# B&R Automation Studio project laba2
Automation Studio 4.5.2.102

## Configuration MainConfig

### Task classes (Cpu.sw)
```
Cyclic#1 (cycle 2000 us, tolerance 0 us):
  ncsdcctrl <- ncsdcctrl.prg
Cyclic#3:
  Program <- Program.prg
DataObjects: Acp10sys
NcDataObjects: acp10etxen <- acp10etxen.dob, gAxis01a <- gAxis01obj.gAxis01a.dob, gAxis01i <- gAxis01obj.gAxis01i.dob
Binaries: TCData, udbdef, ashwd, Role, User, sysconf, ashwac, asfw, arconfig, iomap, Acp10map, acp10cfg
Libraries: Acp10sdc [disabled], sys_lib, Runtime, asstring, Acp10man, Acp10par, NcGlobal, Acp10_MC, brsystem, AsBrStr, DriveLib, astime, fileio, powerlnk, asieccon
```

### Hardware
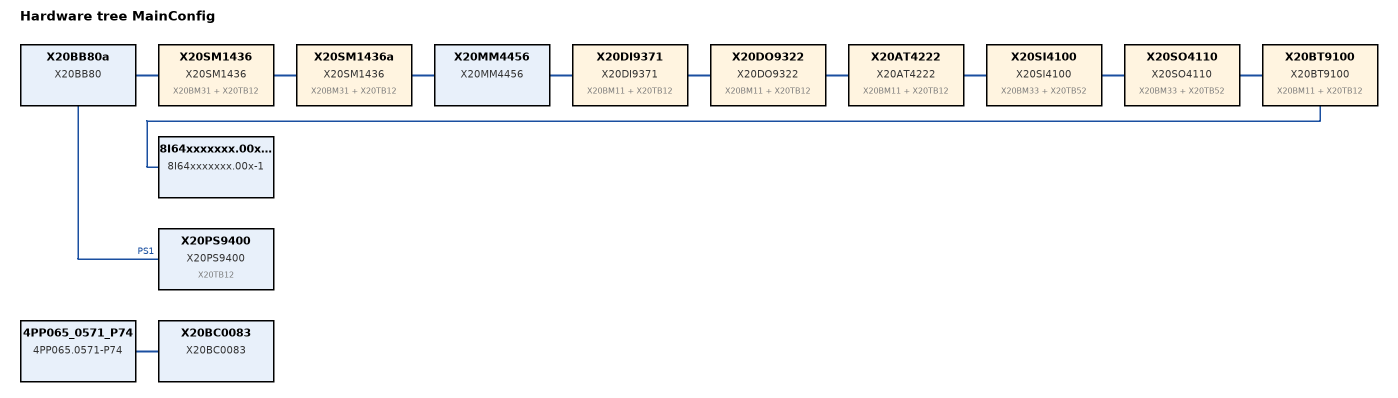
```
4PP065_0571_P74 : 4PP065.0571-P74 v1.1.2.0
  Connector IF4:
    InaNodeNumber = 1
  Connector IF5:
    ActivateDevice = 1
    Mode = Manual
    InternetAddress = 10.0.1.11
    SubnetMask = 255.255.255.0
  ConfigurationID = labBR
  TimerDeviceType = EPLX2X
  TimerDevice = 4PP065_0571_P74.IF4
  TaskClassIdleTime = 2000
  Cyclic1Duration = 2000
  Cyclic1Tolerance = 0
  Cyclic1Output = 1
8I64xxxxxxx.00x-1 : 8I64xxxxxxx.00x-1 v1.3.9.1  [X2X1 -> X20BT9100.X2X1 [Cable Type=X2XCable, Length=10, Version=1.0.0.2]]
  FunctionModel = Standard
  packedETAD = packed
  packedETI = packed
  packedCMDD = packed
  packedCMI = packed
  UNS = 220
  NCR = 10
  NSP = 890
  COS = 64
  RSC = 33000
X20AT4222 : X20AT4222 v1.2.3.0  [SS1 -> X20TB12e.SS; SL -> X20BM11c.SL1]
X20BB80a : X20BB80 v1.0.2.0
X20BC0083 : X20BC0083 v2.14.0.0  [PLK1 -> 4PP065_0571_P74.IF4 (NodeNumber=2) [Cable Type=PowerlinkCable, Length=10, Version=1.0.0.2]; SL -> X20BB80a.SL1]
X20BM11 : X20BM11 v1.0.0.1  [X2X1 -> X20BM33a.X2X2]
X20BM11a : X20BM11 v1.0.0.1  [X2X1 -> X20MM4456.X2X2]
X20BM11b : X20BM11 v1.0.0.1  [X2X1 -> X20BM11a.X2X2]
X20BM11c : X20BM11 v1.0.0.1  [X2X1 -> X20BM11b.X2X2]
X20BM31 : X20BM31 v1.0.0.1  [X2X1 -> X20BB80a.IF1]
X20BM31a : X20BM31 v1.0.0.1  [X2X1 -> X20BM31.X2X2]
X20BM33 : X20BM33 v1.0.0.4  [X2X1 -> X20BM11c.X2X2]
X20BM33a : X20BM33 v1.0.0.4  [X2X1 -> X20BM33.X2X2]
X20BT9100 : X20BT9100 v1.0.3.0  [SS1 -> X20TB12f.SS; SL -> X20BM11.SL1]
X20DI9371 : X20DI9371 v1.0.2.0  [SS1 -> X20TB12c.SS; SL -> X20BM11a.SL1]
X20DO9322 : X20DO9322 v1.0.3.0  [SS1 -> X20TB12d.SS; SL -> X20BM11b.SL1]
X20MM4456 : X20MM4456 v1.4.0.0  [X2X1 -> X20BM31a.X2X2]
X20PS9400 : X20PS9400 v1.0.2.4  [SS1 -> X20TB12.SS; PS -> X20BB80a.PS1]
X20SI4100 : X20SI4100 v1.10.1.1  [SS1 -> X20TB52.SS; SL -> X20BM33.SL1]
X20SM1436 : X20SM1436 v2.3.0.0  [SS1 -> X20TB12a.SS; SL -> X20BM31.SL1]
X20SM1436a : X20SM1436 v2.3.0.0  [SS1 -> X20TB12b.SS; SL -> X20BM31a.SL1]
X20SO4110 : X20SO4110 v1.10.1.1  [SS1 -> X20TB52a.SS; SL -> X20BM33a.SL1]
  SafeModuleID = 3
X20TB12 : X20TB12 v1.0.0.0
X20TB12a : X20TB12 v1.0.0.0
X20TB12b : X20TB12 v1.0.0.0
X20TB12c : X20TB12 v1.0.0.0
X20TB12d : X20TB12 v1.0.0.0
X20TB12e : X20TB12 v1.0.0.0
X20TB12f : X20TB12 v1.0.0.0
X20TB52 : X20TB52 v1.0.0.1
X20TB52a : X20TB52 v1.0.0.1
```

### IoMap.iom - 4PP065_0571_P74/IoMap.iom
```iecst
VAR_CONFIG
	Cyclic#1.gAxis01_DrvIf.iLifeCnt AT %IB."8I64xxxxxxx.00x-1".SDC_LifeCnt;
	Cyclic#1.gAxis01_DrvIf.iDrvOK AT %IX."8I64xxxxxxx.00x-1".ETAD_Input_Bool_02;
	Cyclic#1.gAxis01_DrvIf.oSetTime AT %QW."8I64xxxxxxx.00x-1".SDC_SetTime;
	Cyclic#1.::DoorSM.speed AT %QW."8I64xxxxxxx.00x-1".LFRD_Output;
	Cyclic#1.gAxis01_DiDoIf.iLifeCntDriveReady AT %IB."8I64xxxxxxx.00x-1".SDC_LifeCnt;
	Cyclic#1.gAxis01_DiDoIf.iLifeCntDriveEnable AT %IB."8I64xxxxxxx.00x-1".SDC_LifeCnt;
	Cyclic#1.gAxis01_DiDoIf.oDriveEnable AT %QX."8I64xxxxxxx.00x-1".CMDD_Output_Bool_00;
	Cyclic#1.gAxis01_ModuleOk AT %QX."8I64xxxxxxx.00x-1".CMDD_Output_Bool_01;
	Cyclic#1.gAxis01_ModuleOk AT %QX."8I64xxxxxxx.00x-1".CMDD_Output_Bool_02;
	Cyclic#1.gAxis01_ModuleOk AT %IX."8I64xxxxxxx.00x-1".ModuleOk;
	Cyclic#1.gAxis01_DiDoIf.oDriveEnable AT %QX."8I64xxxxxxx.00x-1".CMDD_Output_Bool_03;
	Cyclic#1.gAxis01_DiDoIf.iDriveReady AT %IX."8I64xxxxxxx.00x-1".ETAD_Input_Bool_02;
	::DriveSM.state AT %IW."8I64xxxxxxx.00x-1".ETAD_Input;
	::DriveSM.command AT %QW."8I64xxxxxxx.00x-1".CMDD_Output;
	::DoorSM.direction AT %IX."X20DI9371".DigitalInput01;
	::DoorSM.sw1 AT %IX."X20DI9371".DigitalInput02;
	::DoorSM.sw2 AT %IX."X20DI9371".DigitalInput03;
	::DoorSM.sw3 AT %IX."X20DI9371".DigitalInput04;
	::DoorSM.sw4 AT %IX."X20DI9371".DigitalInput05;
	::LedSM.led1 AT %QX."X20DO9322".DigitalOutput02;
	::LedSM.led2 AT %QX."X20DO9322".DigitalOutput03;
	::LedSM.led3 AT %QX."X20DO9322".DigitalOutput04;
	::LedSM.led4 AT %QX."X20DO9322".DigitalOutput05;
END_VAR
```

## Logical view

### Global.var
```iecst
VAR
	gAxis01 : ACP10AXIS_typ := (0);
	gAxis01_HW : SdcHwCfg_typ := (0);
	gAxis01_DrvIf : SdcDrvIf16_typ := (0);
	gAxis01_DiDoIf : SdcDiDoIf_typ := (0);
	gAxis01_ModuleOk : BOOL := 0;
	DriveSM : DriveStateMashine := (0);
	DoorSM : DoorStateMashine := (0);
	LedSM : LedStateMashine := (0);
END_VAR
```

### Library Logical/Libraries/DriveLib (ANSIC)

#### Types.typ - Exported data types
```iecst
TYPE
	states_door :
		(
		ST_INIT := 1,
		ST_UNKNOWN := 2,
		ST_OPEN := 3,
		ST_CLOSE := 4,
		ST_ACC_POS := 5,
		ST_ACC_NEG := 6,
		ST_POS := 7,
		ST_NEG := 8,
		ST_DEC_POS := 9,
		ST_DEC_NEG := 10
		);
END_TYPE
```

#### Constants.var - Exported constants
```iecst
VAR CONSTANT
	CMD_ENABLE : USINT := 15;
	CMD_SWITCH_ON : USINT := 7;
	CMD_SHUTDOWN : USINT := 6;
	STATE_DISABLED : USINT := 64;
	STATE_SWITCHED_ON : USINT := 35;
	STATE_READY : USINT := 33;
END_VAR
```

#### DriveLib.fun - Exported functions and function blocks
```iecst
{REDUND_ERROR} FUNCTION_BLOCK DriveStateMashine (*TODO: Add your comment here*) (*$GROUP=User,$CAT=User,$GROUPICON=User.png,$CATICON=User.png*)
	VAR_INPUT
		state : {REDUND_UNREPLICABLE} UINT;
		enable : BOOL;
	END_VAR
	VAR_OUTPUT
		command : UINT;
		speed : INT;
	END_VAR
END_FUNCTION_BLOCK

{REDUND_ERROR} FUNCTION_BLOCK DoorStateMashine (*TODO: Add your comment here*) (*$GROUP=User,$CAT=User,$GROUPICON=User.png,$CATICON=User.png*)
	VAR_INPUT
		state : UINT;
		sw1 : BOOL;
		sw2 : BOOL;
		sw3 : BOOL;
		sw4 : BOOL;
		direction : BOOL;
	END_VAR
	VAR_OUTPUT
		speed : INT;
	END_VAR
END_FUNCTION_BLOCK

{REDUND_ERROR} {REDUND_UNREPLICABLE} FUNCTION_BLOCK LedStateMashine (*TODO: Add your comment here*) (*$GROUP=User,$CAT=User,$GROUPICON=User.png,$CATICON=User.png*)
	VAR_INPUT
		state : {REDUND_UNREPLICABLE} UINT;
	END_VAR
	VAR_OUTPUT
		led1 : {REDUND_UNREPLICABLE} BOOL;
		led2 : {REDUND_UNREPLICABLE} BOOL;
		led3 : {REDUND_UNREPLICABLE} BOOL;
		led4 : {REDUND_UNREPLICABLE} BOOL;
		timer : {REDUND_UNREPLICABLE} INT;
	END_VAR
END_FUNCTION_BLOCK
```

#### DriveStateMashine.c
```c
#include <bur/plctypes.h>
#ifdef __cplusplus
	extern "C"
	{
#endif
	#include "DriveLib.h"
#ifdef __cplusplus
	};
#endif
/* TODO: Add your comment here */
void DriveStateMashine(struct DriveStateMashine* inst)
{
	UINT mask = inst->state & 0x6f;
	if (inst->enable)
	{
		switch (mask)
		{
			case STATE_DISABLED:
				{
					inst->command = CMD_SHUTDOWN;
					break;
				}
			case STATE_READY:
				{
					inst->command = CMD_ENABLE;
					break;
				}
			case STATE_SWITCHED_ON:
				{
					inst->command = CMD_SWITCH_ON;
					break;
				}
		}

	}
	else
	{
		inst->state = STATE_DISABLED;
		inst->command = CMD_SHUTDOWN;
	}

	/*
	DoorSM(&());
	if (!(door->sw1))
	{
		DriveSM.state = STATE_SWITCHED_ON;
	}
	else
	{
		DriveSM.state = STATE_READY;
	}

	if (DriveSM.state == STATE_SWITCHED_ON)
	{
		DriveSM.command = CMD_SWITCH_ON;
	}
	else
	{
		DriveSM.command = CMD_ENABLE;
	}
	*/
}
```

#### DoorStateMashine.c
```c
#include <bur/plctypes.h>
#ifdef __cplusplus
	extern "C"
	{
#endif
	#include "DriveLib.h"
#ifdef __cplusplus
	};
#endif
/* TODO: Add your comment here */
void DoorStateMashine(struct DoorStateMashine* inst)
{
	UINT LOW_SPEED = 100;
	UINT HIGH_SPEED = 200;

	switch(inst->state)
	{

		case ST_INIT:
			{

			/*
				inst->speed = 0;
				if (inst->sw1 == 0 && inst->sw2 == 0 && inst->sw3 == 0 && inst->sw4 == 0)
					inst->state = ST_OPEN;
				else if (inst->sw1 == 1 && inst->sw2 == 1 && inst->sw3 == 1 && inst->sw4 == 1)
				{
					inst->state = ST_CLOSE;
				}
				else
				{
					inst->state = ST_UNKNOWN;
				}

				*/
				inst->state = ST_UNKNOWN;
				break;
			}
		case ST_UNKNOWN:
			{
				/*
				inst->speed = 0;
				if (inst->direction == 1)
				{
					if (inst->sw1 == 0 && inst->sw2 == 0 && inst->sw3 == 0 && inst->sw4 == 0)
						inst->state = ST_OPEN;
					if (inst->sw1 == 1 && inst->sw2 == 0 && inst->sw3 == 0 && inst->sw4 == 0)
						inst->state = ST_ACC_POS;
					if (inst->sw1 == 1 && inst->sw2 == 1 && inst->sw3 == 0 && inst->sw4 == 0)
						inst->state = ST_POS;
					if (inst->sw1 == 1 && inst->sw2 == 1 && inst->sw3 == 1 && inst->sw4 == 0)
						inst->state = ST_DEC_POS;
					if (inst->sw1 == 1 && inst->sw2 == 1 && inst->sw3 == 1 && inst->sw4 == 1)
						inst->state = ST_CLOSE;
				}
				else
				{
					if (inst->sw1 == 1 && inst->sw2 == 1 && inst->sw3 == 1 && inst->sw4 == 1)
						inst->state = ST_CLOSE;
					if (inst->sw1 == 1 && inst->sw2 == 1 && inst->sw3 == 1 && inst->sw4 == 0)
						inst->state = ST_ACC_NEG;
					if (inst->sw1 == 1 && inst->sw2 == 1 && inst->sw3 == 0 && inst->sw4 == 0)
						inst->state = ST_NEG;
					if (inst->sw1 == 1 && inst->sw2 == 0 && inst->sw3 == 0 && inst->sw4 == 0)
						inst->state = ST_DEC_NEG;
					if (inst->sw1 == 0 && inst->sw2 == 0 && inst->sw3 == 0 && inst->sw4 == 0)
						inst->state = ST_OPEN;
				}
				*/
				if (inst->direction == 1)
				{
					inst->speed = 50;
					if (inst->sw4 == 1)
					{
						inst->state = ST_CLOSE;
					}
				}
				else
				{
					inst->speed = -50;
					if (inst->sw1 == 0)
					{
						inst->state = ST_OPEN;
					}
				}
				break;
			}
		case ST_OPEN:
			{
				inst->speed = 0;
				if (inst->direction == 1)
				{
					inst->state = ST_ACC_POS;
				}
				break;
			}
		case ST_ACC_POS:
			{
				inst->speed = LOW_SPEED;
				if (inst->direction == 1 && inst->sw2 == 1)
				{
					inst->state = ST_POS;
				}
				else if (inst->direction == 0)
				{
					inst->state = ST_DEC_NEG;
				}
				break;
			}
		case ST_POS:
			{
				inst->speed = HIGH_SPEED;
				if (inst->direction == 1 && inst->sw3 == 1)
				{
					inst->state = ST_DEC_POS;
				}
				else if (inst->direction == 0)
				{
					inst->state = ST_NEG;
				}
				break;
			}
		case ST_DEC_POS:
			{
				inst->speed = LOW_SPEED;
				if (inst->direction == 1 && inst->sw4 == 1)
				{
					inst->state = ST_CLOSE;
				}

				break;
			}

		case ST_CLOSE:
			{
				inst->speed = 0;
				if (inst->direction == 0)
				{
					inst->state = ST_ACC_NEG;
				}

				break;
			}
		case ST_ACC_NEG:
			{
				inst->speed = -LOW_SPEED;
				if (inst->direction == 0 && inst->sw3 == 0)
				{
					inst->state = ST_NEG;
				}
				else if (inst->direction == 1)
				{
					inst->state = ST_DEC_POS;
				}

				break;
			}
		case ST_NEG:
			{
				inst->speed = -HIGH_SPEED;
				if (inst->direction == 0 && inst->sw2 == 0)
				{
					inst->state = ST_DEC_NEG;
				}
				else if (inst->direction == 1)
				{
					inst->state = ST_POS;
				}

				break;
			}
		case ST_DEC_NEG:
			{
				inst->speed = -LOW_SPEED;
				if (inst->direction == 0 && inst->sw1 == 0)
				{
					inst->state = ST_OPEN;
				}
				break;
			}

	}
}
```

#### LedStateMashine.c
```c
#include <bur/plctypes.h>
#ifdef __cplusplus
	extern "C"
	{
#endif
	#include "DriveLib.h"
#ifdef __cplusplus
	};
#endif
/* TODO: Add your comment here */
void LedStateMashine(struct LedStateMashine* inst)
{
	switch(inst->state)
	{
		case ST_INIT:
			{
				inst->led1 = 0;
				inst->led2 = 0;
				inst->led3 = 0;
				inst->led4 = 0;
				break;
			}
		case ST_UNKNOWN:
			{
				if (inst->timer%21==10)
				{
					inst->led1 = !inst->led1;
					inst->led2 = !inst->led2;
					inst->led3 = !inst->led3;
					inst->led4 = !inst->led4;
				}

				break;
			}
		case ST_OPEN:
			{
				inst->led1 = 0;
				inst->led2 = 0;
				inst->led3 = 0;
				inst->led4 = 0;
				break;
			}
		case ST_ACC_POS:
			{
				inst->led1 = 1;
				if (inst->timer%21 == 10)
				{
					inst->led2 = !inst->led2;
				}
				inst->led3 = 0;
				inst->led4 = 0;
				break;
			}
		case ST_POS:
			{
				inst->led1 = 1;
				inst->led2 = 1;
				if (inst->timer%21 == 10)
				{
					inst->led3 = !inst->led3;
				}
				inst->led4 = 0;
				break;
			}
		case ST_DEC_POS:
			{
				inst->led1 = 1;
				inst->led2 = 1;
				inst->led3 = 1;
				if (inst->timer%21 == 10)
				{
					inst->led4 = !inst->led4;
				}

				break;
			}
		case ST_CLOSE:
			{
				inst->led1 = 1;
				inst->led2 = 1;
				inst->led3 = 1;
				inst->led4 = 1;
				break;
			}
		case ST_ACC_NEG:
			{
				inst->led1 = 1;
				inst->led2 = 1;
				if (inst->timer%21 == 10)
				{
					inst->led3 = !inst->led3;
				}
				inst->led4 = 0;
				break;
			}
		case ST_NEG:
			{
				inst->led1 = 1;
				if (inst->timer%21 == 10)
				{
					inst->led2 = !inst->led2;
				}
				inst->led3 = 0;
				inst->led4 = 0;
				break;
			}
		case ST_DEC_NEG:
			{
				if (inst->timer%21 == 10)
				{
					inst->led1 = !inst->led1;
				}
				inst->led2 = 0;
				inst->led3 = 0;
				inst->led4 = 0;
				break;
			}

	}
	inst->timer++;
}
```

### Program Logical/Program

#### Cyclic.c
```c
#include <bur/plctypes.h>

#ifdef _DEFAULT_INCLUDES
	#include <AsDefault.h>
#endif

void _CYCLIC ProgramCyclic(void)
{

	DoorStateMashine(&DoorSM);
	DriveSM.speed = DoorSM.speed;

	DriveStateMashine(&DriveSM);
	LedSM.state = DoorSM.state;

	LedStateMashine(&LedSM);

	/*
	if (!DoorSM.sw1)
	{
		DriveSM.state = 35;
	}
	else
	{
		DriveSM.state = 33;
	}

	if (DriveSM.state == 35)
	{
		DriveSM.command = 7;
	}
	else
	{
		DriveSM.command = 15;
	}
*/

}
```

#### Init.c
```c
#include <bur/plctypes.h>

#ifdef _DEFAULT_INCLUDES
	#include <AsDefault.h>
#endif

void _INIT ProgramInit(void)
{
	//DoorSM.state = 1;
	//DriveSM.speed = 100;
	//LedSM.led1 = 1;
	//LedSM.led2 = 1;
	//DriveSM.state = 33;
	//DriveSM.command = 6;
	DoorSM.state = 1;
	DriveSM.enable = 1;
}
```
